TYPE st_Firedetection_params :
STRUCT
	r_COwarningLevel_1				: REAL := 10;
	r_COwarningLevel_2				: REAL := 20;
	r_COalarmLevel					: REAL := 120;
	r_COrange						: REAL := 500;
END_STRUCT
END_TYPE

(* stored: Version 1.1.0.1, ProductVersion 3.1.4026.18
   DUT st_Firedetection_params: Id {b4e93580-0161-4c57-a115-e0cd463018f4} *)
